TYPE ST_LinearTable :
STRUCT
	object : AXIS_REF;
	bProx : POINTER TO BOOL;
END_STRUCT
END_TYPE

(* stored: Version 1.1.0.1, ProductVersion 3.1.4026.11
   DUT ST_LinearTable: Id {1fccbdc4-3531-43f0-83a7-157cf626b3cf} *)
